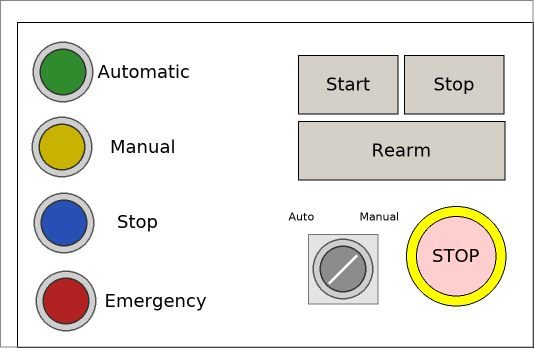
VISUALIZATION MainHMI  // 534x348
    RoundedRectangle (17,22 517x326)
    Lamp1 (28,37 70x70), variable: VisuLogic.L_Run, style: Lamp-Lamp1-Green
    Label (95,57 98x30), "Automatic"
    Label (94,132 98x30), "Manual"
    Lamp1 (27,112 70x70), variable: VisuLogic.L_Manual, style: Lamp-Lamp1-Yellow
    Label (99,207 77x30), "Stop"
    Lamp1 (29,188 70x70), variable: VisuLogic.L_StopOP, style: Lamp-Lamp1-Blue
    Label (98,286 115x30), "Emergency"
    Lamp1 (31,266 70x70), variable: VisuLogic.L_StopEM, style: Lamp-Lamp1-Red
    Rectangle (298,55 100x59), "Start"
        tap HMI.Bt_Run
    Rectangle (404,55 100x59), "Stop"
        tap HMI.Bt_Stop
    Rectangle (298,121 207x59), "Rearm"
        tap HMI.Bt_Rearm
    Ellipse (406,206 100x100)
    Ellipse (416,216 80x80), "STOP"
        toggle HMI.Bt_EmStop
    RotarySwitch (308,234 70x70), variable: HMI.Sel_ManAuto, behaviour: TOGGLE, style: Switch-RotarySwitch-Gray
    Label (283,202 122x30), "Auto Manual"
END_VISUALIZATION

(* stored: Version 1.1.0.1, ProductVersion 3.1.4024.9
   Visu MainHMI: Id {0172a1fd-df4d-437d-8e15-edc9aa511a18} *)
